// TIA Portal V20 export
TYPE "LKinCtrl_typePnPDynamics"
   STRUCT
      path : "LKinCtrl_typePathDynamics";   // Specification of the path dynamics
      orientation : "LKinCtrl_typePathDynamics";   // Specification of the orientation dynamics
      dynamicAdaption : DInt := -1;   // 0=no dynamic adaption, 1=dynamic adaptation with segmentation of the path, 2=dynamic adaptation without segmentation of the path
   END_STRUCT;
END_TYPE
